TEXTLIST TextList_EnvironmentState
  0 = 'ready'
  100 = 'error'
   = ''
END_TEXTLIST

(* stored: Version 1.1.0.1, ProductVersion 3.1.4024.11
   TextList TextList_EnvironmentState: Id {7133280b-a8da-4ae3-bfdb-564ab483c2fc} *)
